(* CoDeSys 2.3.9.62 project: Mezcladora.pro *)
(* Libraries: Standard.lib 2.6.14 11:37:46, IecSfc.lib 2.6.14 12:37:46 *)

(* Task configuration *)
TASK NewTask (PRIORITY := 1, INTERVAL := T#100ms);
	PLC_PRG
END_TASK

(* Global variable list: Global_Variables *)
VAR_GLOBAL
   (* Entradas*)
    LInf: BOOL;
    LSup:BOOL;
    PS1:BOOL;
    PS2:BOOL;
    M:BOOL;
    P:BOOL;
    MV1:BOOL:=FALSE;
    MV2:BOOL:=FALSE;
    MVA:BOOL:=FALSE;
    MVB:BOOL:=FALSE;
    MVC:BOOL:=FALSE;
    MMotor:BOOL:=FALSE;
    Auto:BOOL:=TRUE;

   (*Salidas*)

   Valvula1:BOOL;
   Valvula2:BOOL;
   ValvulaA:BOOL;
   ValvulaB:BOOL;
   ValvulaC:BOOL;
   Motor:BOOL;
   FinAuto:BOOL;
   FinManual:BOOL;

  (* Modos*)
  ON:BOOL;
  Manual:BOOL;
  Automatico:BOOL;
  IniAuto:BOOL;
  IniManual:BOOL;
  Vaciado:BOOL;


END_VAR

(* POU PLC_PRG, ST *)
PROGRAM PLC_PRG
VAR
END_VAR
Depositos;
SelectorModo;
MarchaParada;

IF(IniAuto) THEN
ModoAuto;
END_IF
IF(IniManual) THEN
ModoManual;
END_IF
END_PROGRAM

(* POU Depositos, ST *)
PROGRAM Depositos
VAR
   Nivel: REAL:=0.2;
   ValvulaEntrada:BOOL;
   ValvulaSalida:BOOL;
   CaudalEntrada:REAL:=0;
   CaudalSalida:REAL:=0;
   Area:REAL:=1;
   IntT:REAL:=0.1;
   KEntrada:REAL:=0.3;
   KSalida:REAL:=0.4;
	Neto: REAL;
	Nivellnf:REAL:=0;
	NivelSup:REAL:=2.2;
	CaudalEntrada2: REAL;
	CaudalSalida2: REAL;
	Neto2: REAL;
	Nivel2: REAL;
	Nivellnf2: REAL:=0;
	NivelSup2: REAL:=4;
	KSalida2: REAL:=0.8;
       Texto:STRING;
END_VAR
(*Deposito 1 *)
CaudalEntrada:=BOOL_TO_INT(Valvula1)*KEntrada;
CaudalSalida:=BOOL_TO_INT(Valvula2)*KSalida;
Neto:=(CaudalEntrada-CaudalSalida);
IF (Neto<0AND Nivel>Nivellnf) OR (Neto>0 AND Nivel<NivelSup) THEN
   Nivel:=Nivel+IntT*Neto;
END_IF

IF Nivel>0.33 THEN
   LInf:=TRUE;
ELSE
   LInf:=FALSE;
END_IF

IF Nivel>1.85 THEN
   LSup:=TRUE;
ELSE
   LSup:=FALSE;
END_IF

(*Deposito 2 *)
CaudalEntrada2:=(BOOL_TO_INT(ValvulaA)+BOOL_TO_INT(ValvulaB))*KEntrada;
CaudalSalida2:=BOOL_TO_INT(ValvulaC)*KSalida2;
Neto2:=(CaudalEntrada2-CaudalSalida2);
IF (Neto2<0AND Nivel2>Nivellnf2) OR (Neto2>0 AND Nivel2<NivelSup2) THEN
   Nivel2:=Nivel2+IntT*Neto2;
END_IF


IF Nivel2>2 THEN
   PS1:=TRUE;
ELSE
   PS1:=FALSE;
END_IF

IF Nivel2>3 THEN
   PS2:=TRUE;
ELSE
   PS2:=FALSE;
END_IF

IF Auto THEN
  Texto:='Auto';
ELSE
   Texto:='Manual';
END_IF
END_PROGRAM

(* POU SelectorModo, SFC *)
PROGRAM SelectorModo
VAR
END_VAR
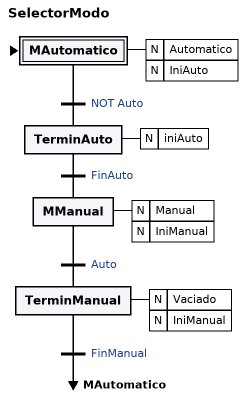
INITIAL_STEP MAutomatico:
	Automatico(N);
	IniAuto(N);
END_STEP
TRANSITION FROM MAutomatico TO TerminAuto := NOT Auto;
END_TRANSITION
STEP TerminAuto:
	iniAuto(N);
END_STEP
TRANSITION FROM TerminAuto TO MManual := FinAuto;
END_TRANSITION
STEP MManual:
	Manual(N);
	IniManual(N);
END_STEP
TRANSITION FROM MManual TO TerminManual := Auto;
END_TRANSITION
STEP TerminManual:
	Vaciado(N);
	IniManual(N);
END_STEP
TRANSITION FROM TerminManual TO MAutomatico := FinManual;
END_TRANSITION
END_PROGRAM

(* POU MarchaParada, SFC *)
PROGRAM MarchaParada
VAR
END_VAR
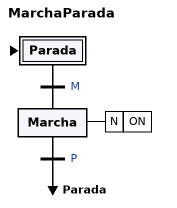
INITIAL_STEP Parada:
END_STEP
TRANSITION FROM Parada TO Marcha := M;
END_TRANSITION
STEP Marcha:
	ON(N);
END_STEP
TRANSITION FROM Marcha TO Parada := P;
END_TRANSITION
END_PROGRAM

(* POU ModoAuto, SFC *)
PROGRAM ModoAuto

VAR
END_VAR
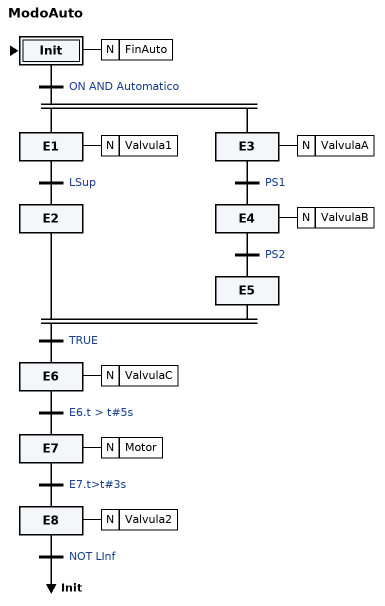
INITIAL_STEP Init:
	FinAuto(N);
END_STEP
TRANSITION FROM Init TO (E1, E3) := ON AND Automatico;
END_TRANSITION
STEP E1:
	Valvula1(N);
END_STEP
TRANSITION FROM E1 TO E2 := LSup;
END_TRANSITION
STEP E2:
END_STEP
STEP E3:
	ValvulaA(N);
END_STEP
TRANSITION FROM E3 TO E4 := PS1;
END_TRANSITION
STEP E4:
	ValvulaB(N);
END_STEP
TRANSITION FROM E4 TO E5 := PS2;
END_TRANSITION
STEP E5:
END_STEP
TRANSITION FROM (E2, E5) TO E6 := TRUE;
END_TRANSITION
STEP E6:
	ValvulaC(N);
END_STEP
TRANSITION FROM E6 TO E7 := E6.t > t#5s;
END_TRANSITION
STEP E7:
	Motor(N);
END_STEP
TRANSITION FROM E7 TO E8 := E7.t>t#3s;
END_TRANSITION
STEP E8:
	Valvula2(N);
END_STEP
TRANSITION FROM E8 TO Init := NOT LInf;
END_TRANSITION
END_PROGRAM

(* POU ModoManual, SFC *)
PROGRAM ModoManual
VAR
END_VAR
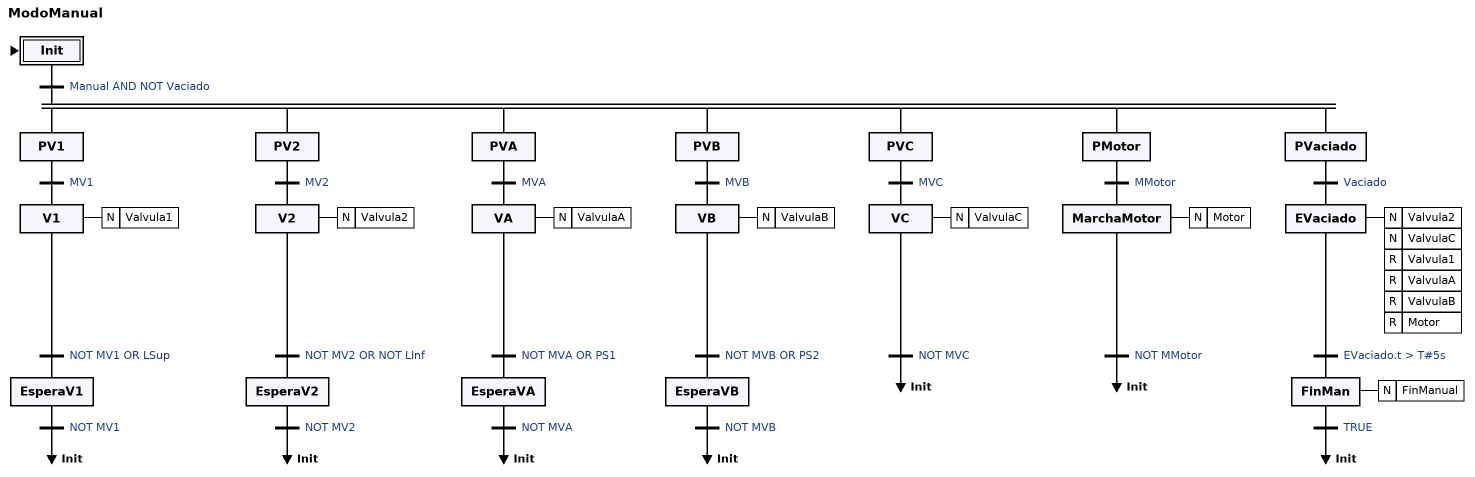
INITIAL_STEP Init:
END_STEP
TRANSITION FROM Init TO (PV1, PV2, PVA, PVB, PVC, PMotor, PVaciado) := Manual AND NOT Vaciado;
END_TRANSITION
STEP PV1:
END_STEP
TRANSITION FROM PV1 TO V1 := MV1;
END_TRANSITION
STEP V1:
	Valvula1(N);
END_STEP
TRANSITION FROM V1 TO EsperaV1 := NOT MV1 OR LSup;
END_TRANSITION
STEP EsperaV1:
END_STEP
TRANSITION FROM EsperaV1 TO Init := NOT MV1;
END_TRANSITION
STEP PV2:
END_STEP
TRANSITION FROM PV2 TO V2 := MV2;
END_TRANSITION
STEP V2:
	Valvula2(N);
END_STEP
TRANSITION FROM V2 TO EsperaV2 := NOT MV2 OR NOT LInf;
END_TRANSITION
STEP EsperaV2:
END_STEP
TRANSITION FROM EsperaV2 TO Init := NOT MV2;
END_TRANSITION
STEP PVA:
END_STEP
TRANSITION FROM PVA TO VA := MVA;
END_TRANSITION
STEP VA:
	ValvulaA(N);
END_STEP
TRANSITION FROM VA TO EsperaVA := NOT MVA OR PS1;
END_TRANSITION
STEP EsperaVA:
END_STEP
TRANSITION FROM EsperaVA TO Init := NOT MVA;
END_TRANSITION
STEP PVB:
END_STEP
TRANSITION FROM PVB TO VB := MVB;
END_TRANSITION
STEP VB:
	ValvulaB(N);
END_STEP
TRANSITION FROM VB TO EsperaVB := NOT MVB OR PS2;
END_TRANSITION
STEP EsperaVB:
END_STEP
TRANSITION FROM EsperaVB TO Init := NOT MVB;
END_TRANSITION
STEP PVC:
END_STEP
TRANSITION FROM PVC TO VC := MVC;
END_TRANSITION
STEP VC:
	ValvulaC(N);
END_STEP
TRANSITION FROM VC TO Init := NOT MVC;
END_TRANSITION
STEP PMotor:
END_STEP
TRANSITION FROM PMotor TO MarchaMotor := MMotor;
END_TRANSITION
STEP PVaciado:
END_STEP
TRANSITION FROM PVaciado TO EVaciado := Vaciado;
END_TRANSITION
STEP EVaciado:
	Valvula2(N);
	ValvulaC(N);
	Valvula1(R);
	ValvulaA(R);
	ValvulaB(R);
	Motor(R);
END_STEP
TRANSITION FROM EVaciado TO FinMan := EVaciado.t > T#5s;
END_TRANSITION
STEP FinMan:
	FinManual(N);
END_STEP
TRANSITION FROM FinMan TO Init := TRUE;
END_TRANSITION
STEP MarchaMotor:
	Motor(N);
END_STEP
TRANSITION FROM MarchaMotor TO Init := NOT MMotor;
END_TRANSITION
END_PROGRAM

(* Visualisation Deposito
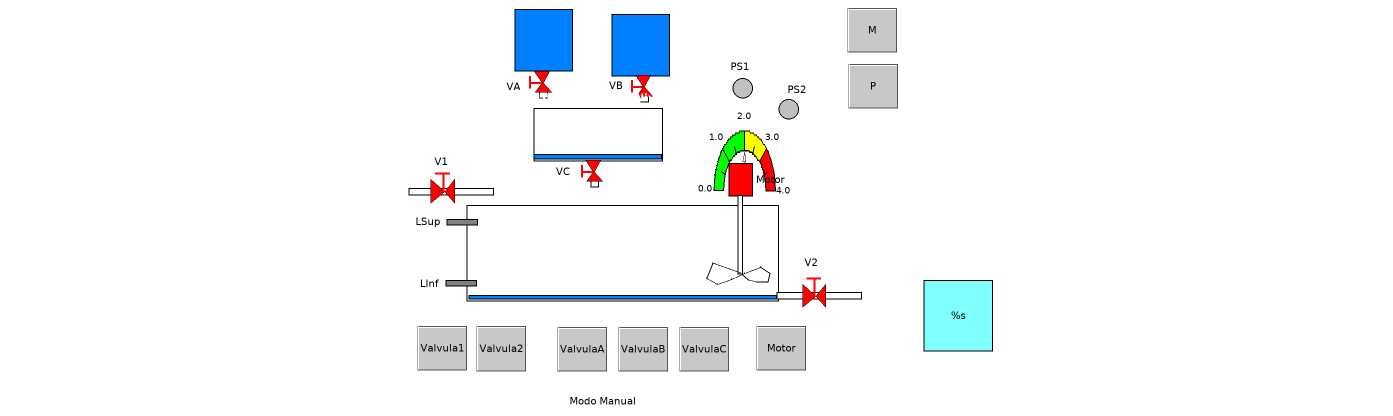
button at (30,345)-(79,389): text "Valvula1"; toggles MV1
button at (89,345)-(138,390): text "Valvula2"; toggles MV2
rectangle at (81,314)-(389,318): top -40*Depositos.Nivel
rectangle at (389,311)-(474,318): alarm colour if Valvula2 AND Depositos.Nivel>0
rectangle at (21,207)-(106,214): alarm colour if Valvula1
group at (43,192)-(67,222)
  polygon at (0,6)-(13,29): alarm colour if Valvula1
  polygon at (13,6)-(23,29): alarm colour if Valvula1
  polyline at (12,0)-(12,17): alarm colour if Valvula1
  polyline at (4,0)-(18,0): alarm colour if Valvula1
polygon at (415,303)-(428,326): alarm colour if Valvula2
polygon at (428,303)-(438,326): alarm colour if Valvula2
polyline at (427,297)-(427,314): alarm colour if Valvula2
polyline at (419,297)-(433,297): alarm colour if Valvula2
rectangle at (59,238)-(90,244): alarm colour if LSup
rectangle at (58,299)-(89,305): alarm colour if LInf
group at (142,90)-(164,117)
  polygon at (4,0)-(19,11): alarm colour if ValvulaA
  polygon at (5,11)-(21,21): alarm colour if ValvulaA
  polyline at (0,12)-(11,12): alarm colour if ValvulaA
  polyline at (0,5)-(0,17): alarm colour if ValvulaA
polygon at (248,94)-(263,105): alarm colour if ValvulaB
polygon at (249,105)-(265,115): alarm colour if ValvulaB
polyline at (244,106)-(255,106): alarm colour if ValvulaB
polyline at (244,99)-(244,111): alarm colour if ValvulaB
button at (170,346)-(219,390): text "ValvulaA"; toggles MVA
button at (231,346)-(280,390): text "ValvulaB"; toggles MVB
polygon at (198,179)-(213,190): alarm colour if ValvulaC
polygon at (199,190)-(215,200): alarm colour if ValvulaC
polyline at (194,191)-(205,191): alarm colour if ValvulaC
polyline at (194,184)-(194,196): alarm colour if ValvulaC
button at (292,346)-(341,390): text "ValvulaC"; toggles MVC
rectangle at (146,173)-(274,178): top -10*Depositos.Nivel2
group at (308,116)-(405,223)
  rectangle at (0,0)-(1,1): text "{ExtendedElement},Visu\ElementDLL.ete,0,@Zeigerinstrument,97,180,0,0,255,255,255,0,Depositos.Nivel2,,%.1f,0,1,1,0.5,1,0,4,0,0,0,0,0,0,0,-11,80,400,Arial,1,3,0,2,0,255,0,2,3,255,255,0,3,4,255,0,0,0,255,255,255,,0,0,0,0,"
  rectangle at (0,41)-(19,55): text "0.0"
  rectangle at (11,14)-(30,28): text "1.0"
  rectangle at (39,3)-(58,17): text "2.0"
  rectangle at (67,14)-(86,28): text "3.0"
  rectangle at (78,42)-(97,56): text "4.0"
  polygon at (47,29)-(50,49): angle ((Depositos.Nivel2 * 1.0)-2) * 45
ellipse at (345,97)-(365,117): alarm colour if PS1
ellipse at (391,118)-(411,138): alarm colour if PS2
rectangle at (35,165)-(72,196): text "V1"
rectangle at (405,266)-(442,297): text "V2"
rectangle at (107,90)-(144,121): text "VA"
rectangle at (210,89)-(247,120): text "VB"
rectangle at (157,175)-(194,206): text "VC"
rectangle at (334,70)-(371,101): text "PS1"
rectangle at (391,93)-(428,124): text "PS2"
rectangle at (23,287)-(60,318): text "LInf"
rectangle at (22,225)-(59,256): text "LSup"
rectangle at (341,182)-(365,215): alarm colour if Motor
rectangle at (364,183)-(401,214): text "Motor"
button at (460,27)-(509,71): text "M"; taps M
button at (369,345)-(418,389): text "Motor"; toggles MMotor
rectangle at (168,400)-(262,440): text "Modo Manual"
button at (461,83)-(510,127): text "P"; taps P
rectangle at (536,299)-(605,370): text "%s"; shows Depositos.Texto; alarm colour if Auto; toggles Auto
25 more shapes without text or variables
*)
